TYPE ST_AdsAdress :
STRUCT
	sNetId	: STRING(23);
	nPort	: UINT;
END_STRUCT
END_TYPE

(* stored: Version 1.1.0.1, ProductVersion 3.1.0.23
   DUT ST_AdsAdress: Id {27df2324-8b2b-4173-ad01-a372b297f9a3} *)
